Staubli VAL3: OnEvent12.pgx

program OnEvent12()
begin
  //-----------------------------------------------------------------------
  //Header begin
  //LasMAN3.7
  //Description of program
  //
  //Input parameters
  //
  //Output paramaters
  //Example
  //  call OnEvent1()
  //History
  //  Creation : 2013-06-23  y.ye@staubli.com
  //Header end
  //-----------------------------------------------------------------------
  resetMotion()
  if TxtFile:b7Axis
    // call Teach:Teach7Axis(TxtFile:trAxisData.x,TxtFile:trAxisData.y,0)
    call Teach:TeachAxis(TxtFile:trAxisData.x,TxtFile:trAxisData.y,TxtFile:trAxisData.z,TxtFile:trAxisData.rx,false)
  else
    popUpMsg("请到选项界面中激活七轴")
  endIf
  DataBase:nInterfaceType=9
end
